ABB RAPID module: MainModule.mod

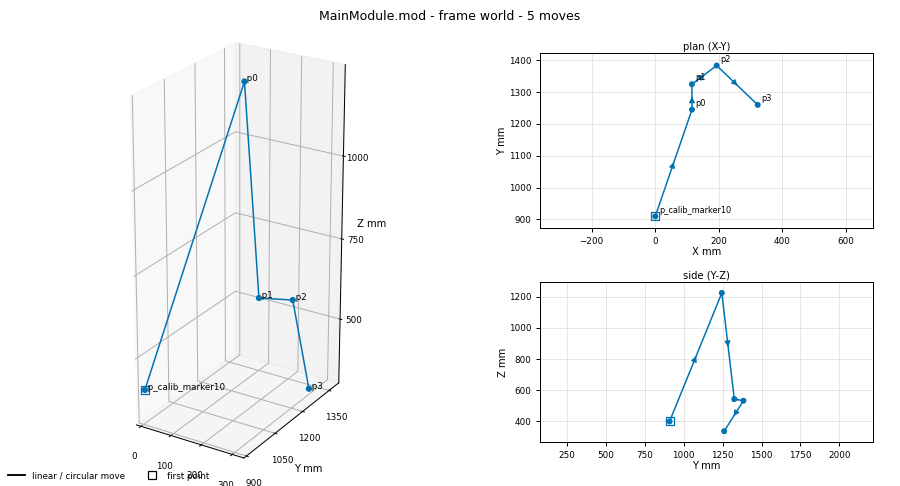
[picture p0: tool path of MainModule.mod in frame world, 5 of 6 moves have a stored position in this frame; points joined in program order, loops and branches not executed]
MODULE MainModule
	CONST robtarget p1:=[[115.36,1324.97,543.37],[0.259423,-0.956125,-0.0586915,0.122802],[0,-1,0,1],[9E+09,9E+09,9E+09,9E+09,9E+09,9E+09]];
	PERS tooldata photoneo:=[TRUE,[[-83.9293,104.623,159.994],[0.703963,-0.268575,0.100635,-0.649751]],[0.3,[0,0,160],[1,0,0,0],0,0,0]];
	CONST robtarget p0:=[[115.50,1244.97,1224.88],[0.471132,-0.873001,-0.0527845,0.114531],[0,-1,0,1],[9E+09,9E+09,9E+09,9E+09,9E+09,9E+09]];
	CONST robtarget p2:=[[193.16,1383.71,532.81],[0.267706,-0.816352,-0.49286,0.137812],[0,-2,0,1],[9E+09,9E+09,9E+09,9E+09,9E+09,9E+09]];
	CONST robtarget p11:=[[193.16,1383.71,532.81],[0.267706,-0.816351,-0.492861,0.137811],[0,-2,0,1],[9E+09,9E+09,9E+09,9E+09,9E+09,9E+09]];
	LOCAL PERS robtarget p_calib_marker:=[[-505.87,1375.53,432.56],[0.493544,-0.492667,-0.506267,-0.507334],[1,0,-3,1],[9E+09,9E+09,9E+09,9E+09,9E+09,9E+09]];
	CONST robtarget p10:=[[-505.87,1375.53,432.56],[0.493544,-0.492666,-0.506266,-0.507335],[1,0,-3,1],[9E+09,9E+09,9E+09,9E+09,9E+09,9E+09]];
	CONST robtarget p_calib_marker10:=[[0.11,909.30,399.58],[0.500728,-0.499662,0.499327,0.500282],[0,-1,-1,1],[9E+09,9E+09,9E+09,9E+09,9E+09,9E+09]];
	LOCAL CONST jointtarget jposhome:=[[77.5626,5.48013,1.9853,-70.0348,-13.2221,69.1978],[9E+09,9E+09,9E+09,9E+09,9E+09,9E+09]];
	CONST robtarget p20:=[[115.52,1244.97,1224.86],[0.471123,-0.87301,-0.0528002,0.114491],[0,-1,0,1],[9E+09,9E+09,9E+09,9E+09,9E+09,9E+09]];
	LOCAL PERS robtarget p3:=[[322.31,1259.93,336.95],[0.475534,-0.693661,-0.431801,0.325959],[0,-1,0,1],[9E+09,9E+09,9E+09,9E+09,9E+09,9E+09]];
	CONST robtarget p12:=[[322.31,1259.93,336.95],[0.475535,-0.693661,-0.4318,0.32596],[0,-1,0,1],[9E+09,9E+09,9E+09,9E+09,9E+09,9E+09]];
	PROC main()
		MoveAbsJ jposhome\NoEOffs, v100, z50, photoneo;
		!MoveL p0, v100, z50, photoneo;
		MoveL p_calib_marker10, v50, z0, tool0;
		MoveL p0, v100, z50, photoneo;
		MoveL p1, v100, z50, photoneo;
		MoveL p2, v100, z50, photoneo;
		MoveL p3, v100, z50, photoneo;
	ENDPROC
ENDMODULE
